{attribute 'qualified_only'}
TYPE ENUM_XPIM_Filters :
(
    Unknown := 0,
    T50 := 1,
    T25 := 2,
    T10 := 3,
    T5 := 4,
    T1 := 5,
    T100 := 6
);
END_TYPE

(* stored: Version 1.1.0.1
   DUT ENUM_XPIM_Filters: Id {bfdc46b8-f018-4652-86e1-1c12b2ad37bb} *)
